DATA_BLOCK "ST10_FB_Tower_4Lamp_DB"
{ S7_Optimized_Access := 'TRUE' }
VERSION : 0.1
NON_RETAIN
// ATTRIBUTES
// AUTO_NUMBER = False
// BLOCK_NUMBER = 5050
// END_ATTRIBUTES
"FB_Tower_4Lamp"

BEGIN

END_DATA_BLOCK

